(* CODESYS project Uppgift14.project

Project tree, tasks and I/O mapping:
  Device : CODESYS Control Win V3, 3S - Smart Software Solutions GmbH, order no. 305021, version 3.5.10.40
    application Application
      libraries: Standard, * (System)
      task MainTask (cyclic, interval t#20ms, priority 1) calls PLC_PRG
      program PLC_PRG [SFC]: PackageToDoor, OpenDoorTask, MoveObjectThroueDoor, CloseDoorTask, ResetMotor, ResetEngene2, BlinkingLights
      global variables GVL
      Symbols
*)

// Device/Application/GVL
{attribute 'qualified_only'}
VAR_GLOBAL
	Sensor1: BOOL;
	Sensor2: BOOL;
	Sensor3:  BOOL;
	SensorClose: BOOL;
	SensorOpen: BOOL;
	
	Conv1MotorFwd: BOOL;
	Conv2MotorFwd: BOOL;
	DoorMotorFwd: BOOL;
	DoorMotorRev: BOOL;
	Light: BOOL;
END_VAR

// Device/Application/PLC_PRG
PROGRAM PLC_PRG
VAR
	
	OutTime: TIME;
	OutTime2: TIME;
	LightTimerOFf: TOF;
	LightTimeOn: TON;
END_VAR
VAR // added by the converter: edge detectors and wires of the graphical bodies
    _w1, _w2, _w4, _w5, _w6, _w8, _w9 : ANY;
    _w3, _w7 : BOOL;
END_VAR

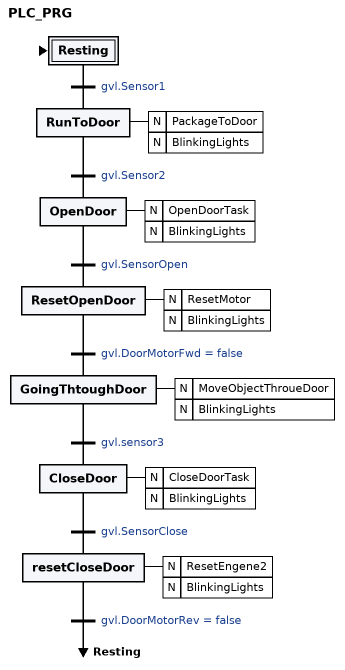
INITIAL_STEP Resting:
END_STEP
TRANSITION FROM Resting TO RunToDoor
    := gvl.Sensor1;
END_TRANSITION
STEP RunToDoor:
    PackageToDoor(N);
    BlinkingLights(N);
END_STEP
TRANSITION FROM RunToDoor TO OpenDoor
    := gvl.Sensor2;
END_TRANSITION
STEP OpenDoor:
    OpenDoorTask(N);
    BlinkingLights(N);
END_STEP
TRANSITION FROM OpenDoor TO ResetOpenDoor
    := gvl.SensorOpen;
END_TRANSITION
STEP ResetOpenDoor:
    ResetMotor(N);
    BlinkingLights(N);
END_STEP
TRANSITION FROM ResetOpenDoor TO GoingThtoughDoor
    := gvl.DoorMotorFwd = false;
END_TRANSITION
STEP GoingThtoughDoor:
    MoveObjectThroueDoor(N);
    BlinkingLights(N);
END_STEP
TRANSITION FROM GoingThtoughDoor TO CloseDoor
    := gvl.sensor3;
END_TRANSITION
STEP CloseDoor:
    CloseDoorTask(N);
    BlinkingLights(N);
END_STEP
TRANSITION FROM CloseDoor TO resetCloseDoor
    := gvl.SensorClose;
END_TRANSITION
STEP resetCloseDoor:
    ResetEngene2(N);
    BlinkingLights(N);
END_STEP
TRANSITION FROM resetCloseDoor TO Resting
    := gvl.DoorMotorRev = false;
END_TRANSITION

ACTION PackageToDoor:
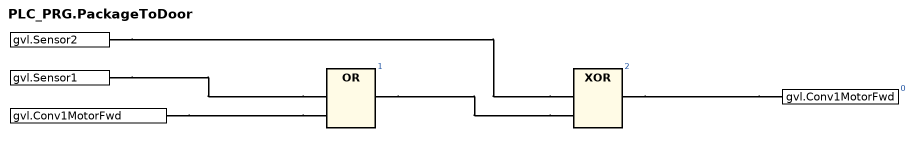
gvl.Conv1MotorFwd := _w1;
_w1 := gvl.Sensor2 XOR (gvl.Sensor1 OR gvl.Conv1MotorFwd);
END_ACTION

ACTION OpenDoorTask:
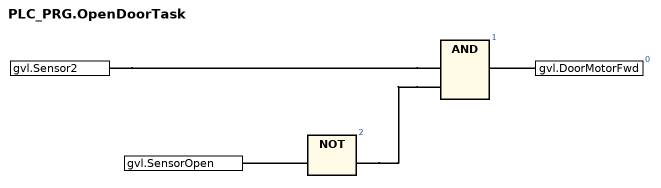
gvl.DoorMotorFwd := _w2;
_w2 := gvl.Sensor2 AND _w3;
_w3 := NOT gvl.SensorOpen;
END_ACTION

ACTION MoveObjectThroueDoor:
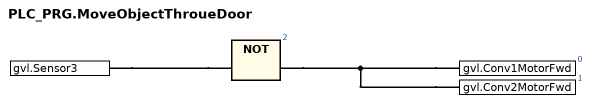
gvl.Conv1MotorFwd := _w4;
gvl.Conv2MotorFwd := _w4;
_w4 := NOT gvl.Sensor3;
END_ACTION

ACTION CloseDoorTask:
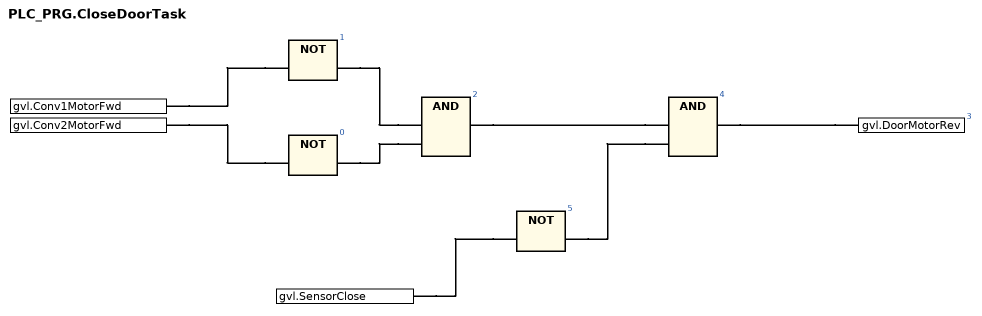
_w5 := NOT gvl.Conv1MotorFwd AND NOT gvl.Conv2MotorFwd;
gvl.DoorMotorRev := _w6;
_w6 := _w5 AND _w7;
_w7 := NOT gvl.SensorClose;
END_ACTION

ACTION ResetMotor:
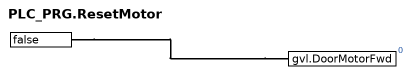
gvl.DoorMotorFwd := false;
END_ACTION

ACTION ResetEngene2:
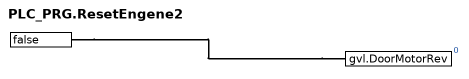
gvl.DoorMotorRev := false;
END_ACTION

ACTION BlinkingLights:
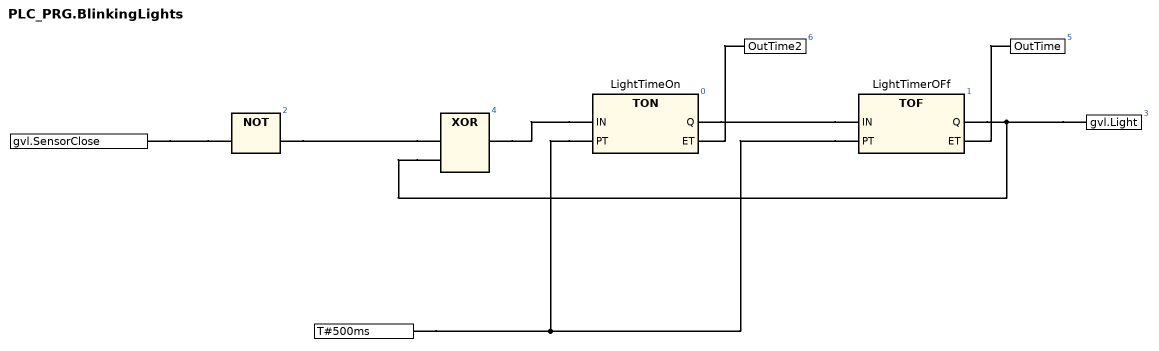
LightTimeOn(IN := _w8, PT := T#500ms); // TON
LightTimerOFf(IN := LightTimeOn.Q, PT := T#500ms); // TOF
_w9 := NOT gvl.SensorClose;
gvl.Light := LightTimerOFf.Q;
_w8 := _w9 XOR LightTimerOFf.Q;
OutTime := LightTimerOFf.ET;
OutTime2 := LightTimeOn.ET;
END_ACTION

END_PROGRAM
